FUNCTION_BLOCK AX_T_FF_SR_SYM_STORE (* Event-driven bistable and Toggle, symmetric Start-Up Behaviour and INIT *)
  (* Standard: 61499-1 Annex A; Description: Copyright (c) 2017 fortiss GmbH, HR Agrartechnik GmbH This program and the accompanying materials are made available under the terms of the Eclipse Public License 2.0 which is available at https://www.eclipse.org/legal/epl-2.0/ SPDX-License-Identifier: EPL-2.0 *)
  (* Version 3.0, 2025-04-14, Patrick Aigner, changed package *)
  (* Version 1.1, 2024-08-27, Franz Höpfinger, HR Agrartechnik GmbH, Copy E_SR and make this FB *)
  (* Version 1.0, 2017-09-22, Alois Zoitl, fortiss GmbH, initial API and implementation and/or initial documentation *)
  PACKAGE adapter::events::unidirectional;
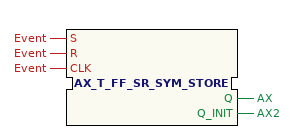
  EVENT_INPUT
    S; (* Set output Q *)
    R; (* Reset output Q *)
    CLK; (* Clock for triggering a output toggle *)
  END_EVENT
  PLUGS
    Q : adapter::types::unidirectional::AX; (* value of flip flop *)
    Q_INIT : adapter::types::bidirectional::AX2; (* Value of Q at INIT *)
  END_PLUGS
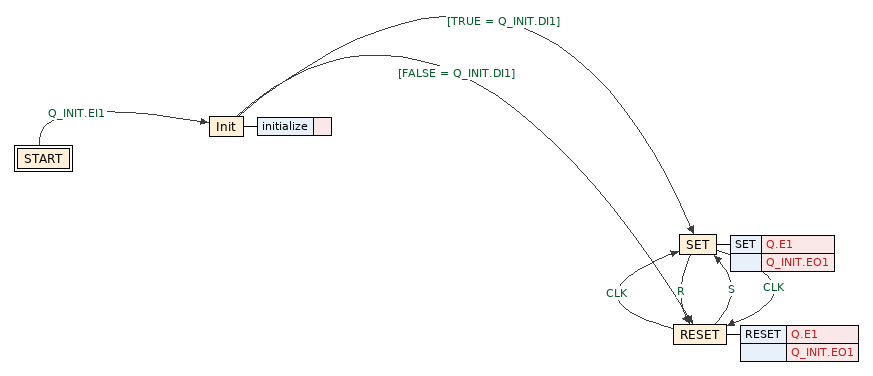
  EC_STATES
    START; (* Initial State *)
    Init : initialize; (* Initialization *)
    SET : SET -> Q.E1, -> Q_INIT.EO1;
    RESET : RESET -> Q.E1, -> Q_INIT.EO1;
  END_STATES
  EC_TRANSITIONS
    SET TO RESET := R;
    RESET TO SET := S;
    SET TO RESET := CLK;
    RESET TO SET := CLK;
    START TO Init := Q_INIT.EI1;
    Init TO RESET := [FALSE = Q_INIT.DI1];
    Init TO SET := [TRUE = Q_INIT.DI1];
  END_TRANSITIONS
  ALGORITHM SET IN ST: (* SET algorithm *)
Q.D1 := TRUE;
Q_INIT.DO1 := TRUE;
  END_ALGORITHM
  ALGORITHM RESET IN ST: (* RESET algorithm *)
Q.D1 := FALSE;
Q_INIT.DO1 := FALSE;
  END_ALGORITHM
END_FUNCTION_BLOCK
